{attribute addProperty BoxType "EPP6090-0000-0017"}
{attribute addProperty Id "DIS_InputsAT %I*DIS_Inputs_23B85B6E1620DIS_OutputsAT %Q*DIS_Outputs_1C156EA83240WcStateAT %I*WcState_F855686C1620InfoDataAT %I*InfoData_BC63D37F80100"}
{attribute addProperty CRC "154045306"}
{attribute addProperty SizeInBites "144"}
{attribute addProperty SizeInBytes "18"}
TYPE EPP6090_C46C03A8 :
STRUCT
	{attribute addProperty Name "DIS_Inputs"}
	DIS_Inputs : DIS_Inputs_23B85B6E;
	{attribute addProperty Name "DIS_Outputs"}
	DIS_Outputs : DIS_Outputs_1C156EA8;
	{attribute addProperty Name "WcState"}
	WcState : WcState_F855686C;
	{attribute addProperty Name "InfoData"}
	InfoData : InfoData_BC63D37F;
END_STRUCT
END_TYPE

(* stored: Version 1.2.0.0, ProductVersion 3.1.4024.9
   DUT EPP6090_C46C03A8: Id {9b6cac2e-5263-4aad-80ba-0ebd9889927f} *)
